{attribute 'strict'}
TYPE E_CognexCameraGetOnlineStatus :
(
	WAITING_FOR_STATUS_CODE								:= 2,
	THE_IN_SIGHT_VISION_SYSTEM_IS_CURRENTLY_OFFLINE		:= 0,
	THE_IN_SIGHT_VISION_SYSTEM_IS_CURRENTLY_ONLINE 		:= 1
);
END_TYPE

(* stored: Version 1.1.0.1, ProductVersion 3.1.4024.12
   DUT E_CognexCameraGetOnlineStatus: Id {bd9faf2f-aef6-462d-8aac-78b048afb531} *)
